{attribute addProperty BoxType "EPP1322-0001-0016"}
{attribute addProperty Id "A_0020_EPP1322_0001_0017A_0020_EPP1322_0001_0017_AE45DA7A2662332.75"}
{attribute addProperty CRC "488834451"}
{attribute addProperty SizeInBites "2662"}
{attribute addProperty SizeInBytes "332.75"}
TYPE A_0019_EPP1322_0001_0016_1D230593 EXTENDS EPP1322_179A0949 :
STRUCT
	{attribute addProperty Name "A_0020_EPP1322_0001_0017"}
	A_0020_EPP1322_0001_0017 : A_0020_EPP1322_0001_0017_AE45DA7A;
END_STRUCT
END_TYPE

(* stored: Version 1.2.0.0, ProductVersion 3.1.4024.9
   DUT A_0019_EPP1322_0001_0016_1D230593: Id {bb1f0ec4-b1dc-4f85-ae43-909439a9f84a} *)
